// TIA Portal project "Drehgeber_0" (V20)

(* hardware
DEVICE "S7-1500/ET200MP-Station_1"  S7-1500 station
   slot 0: "Profilschiene_0"  Rack  6ES7 590-1***0-0AA0
   slot 1: "PLC_1"  CPU 1513-1 PN  6ES7 513-1AM03-0AB0  V4.0
      slot 3: "CPU-Display_1"  6ES7591-1AA00-0AA0
      slot 32768: "PROFINET-Schnittstelle_1"  X1
         slot 32769: "Port_1"  X1 P1
         slot 32770: "Port_2"  X1 P2
      slot 34817: "Virtual CP interface port_1"  Virtual CP interface port  Virtual CP interface port FW V4.0
   slot 2: "DI 16x24VDC BA_1"  DI 16x24VDC BA  6ES7 521-1BH10-0AA0  V1.1
   slot 3: "DQ 16x24VDC/0.5A ST_1"  DQ 16x24VDC/0.5A ST  6ES7 522-1BH00-0AB0  V2.0
   slot 4: "AI 8xU/I/R/RTD BA_2"  AI 8xU/I/R/RTD BA  6ES7 531-7QF00-0AB0  V1.0
   slot 5: "AQ 8xU/I HS_2"  AQ 8xU/I HS  6ES7 532-5HF00-0AB0  V2.2
*)

// ===== PLC "PLC_1"  CPU 1513-1 PN =====

VAR_GLOBAL   // PLC tag table "Eingaenge"
   "1B1" AT %I0.0 : Bool;   // Lichttaster
   "2B1" AT %I0.1 : Bool;   // Drehgeber (Signal A)
   "2B2" AT %I0.2 : Bool;   // Drehgeber (Signal B)
   "3B1" AT %E0.3 : Bool;   // Pusher 1 (hinten)
   "3B2" AT %E0.4 : Bool;   // Pusher 1 (vorne)
   "4B1" AT %E0.5 : Bool;   // Pusher 2 (hinten)
   "4B2" AT %E0.6 : Bool;   // Pusher 2 (vorne)
   "1B2" AT %ED30 : DInt;   // Sichtsensor
END_VAR

VAR_GLOBAL   // PLC tag table "Ausgaenge"
   "1M1" AT %Q0.1 : Bool;   // Förderband (vor)
   "1M2" AT %Q0.2 : Bool;   // Förderband (zurück)
   "3M1" AT %A0.3 : Bool;   // Pusher 1
   "4M1" AT %A0.5 : Bool;   // Pusher 2
END_VAR

DATA_BLOCK "Datenbaustein_1"   // DB1
{ S7_Optimized_Access := 'TRUE' }
VERSION : 0.1
   VAR
      Betriebsdaten : Struct
         Trigger : Struct
            Kanal_A : Struct
               Pos : Bool;
               Neg : Bool;
            END_STRUCT;
            Kanal_B : Struct
               Pos : Bool;
               Neg : Bool;
            END_STRUCT;
         END_STRUCT;
         Drehrichtung : Struct
            Vor : Bool;
            Zurueck : Bool;
         END_STRUCT;
         Pusher : Array[1..2] of Struct
            ID : UDInt;
            Pos_Register : DInt;
            Bauteil_Farbe : Array[0..1] of DInt;
            Zustand : Bool;
            PTRIG : Bool;
         END_STRUCT;
         Geberwert : DInt;
         Position_cm : Real;
         Schieben : Bool;
      END_STRUCT;
   END_VAR
BEGIN
   Betriebsdaten.Pusher[1].Pos_Register := 132;
   Betriebsdaten.Pusher[2].Pos_Register := 210;
END_DATA_BLOCK

DATA_BLOCK "Drehgeber_Signale_DB"   // DB2
{ S7_Optimized_Access := 'TRUE' }
VERSION : 0.1
// stored: InstanceOfName Drehgeber_Signale_Hohe_Aufloesung
"Drehgeber_Signale_Hohe_Aufloesung"
BEGIN
END_DATA_BLOCK

DATA_BLOCK "Schieberegister"   // DB3
{ S7_Optimized_Access := 'TRUE' }
VERSION : 0.1
   VAR
      Aktuelles_Bauteil : DInt;
      Register : Array[0..255] of DInt;
   END_VAR
BEGIN
END_DATA_BLOCK

FUNCTION_BLOCK "Drehgeber_Signale_Hohe_Aufloesung"   // FB1, FBD
{ S7_Optimized_Access := 'TRUE' }
VERSION : 0.1
   VAR
      Laufband_Richtung_DB : "Laufband_Richuntgserkennung";
   END_VAR
BEGIN

REGION Network 1
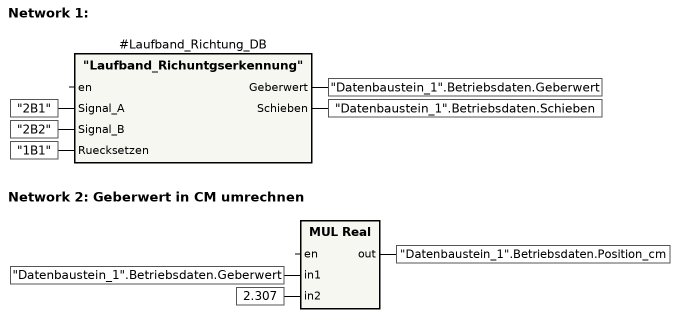
   #Laufband_Richtung_DB(Signal_A := "2B1",   // "Laufband_Richuntgserkennung"
                         Signal_B := "2B2",
                         Ruecksetzen := "1B1",
                         Geberwert => "Datenbaustein_1".Betriebsdaten.Geberwert,
                         Schieben => "Datenbaustein_1".Betriebsdaten.Schieben);
END_REGION

REGION Network 2: Geberwert in CM umrechnen
   "Datenbaustein_1".Betriebsdaten.Position_cm := "Datenbaustein_1".Betriebsdaten.Geberwert * 2.307;
END_REGION
END_FUNCTION_BLOCK

FUNCTION_BLOCK "Laufband_Richuntgserkennung"   // FB2, FBD
{ S7_Optimized_Access := 'TRUE' }
VERSION : 0.1
   VAR_INPUT
      Signal_A : Bool;
      Signal_B : Bool;
      Ruecksetzen : Bool;
   END_VAR
   VAR_OUTPUT
      Geberwert : DInt;
      Schieben : Bool;
   END_VAR
   VAR
      PTRIG_KanalA : Bool;
      NTRIG_KanalA : Bool;
      PTRIG_KanalB : Bool;
      NTRIG_KanalB : Bool;
      PTRIG_SignalA : Bool;
      PTRIG_SignalB : Bool;
      Vor : Bool;
      Zurueck : Bool;
   END_VAR
   VAR_TEMP   // added for the SCL form of the ladder/FBD networks
      _w1 : Bool;
      _w2 : Bool;
      _w3 : Bool;
      _w4 : Bool;
      _w5 : Bool;
   END_VAR
BEGIN

REGION Network 1: Vorwärts
   // Wenn eine positive Flanke von A kommt, wenn B bereits da ist = Vorwärts
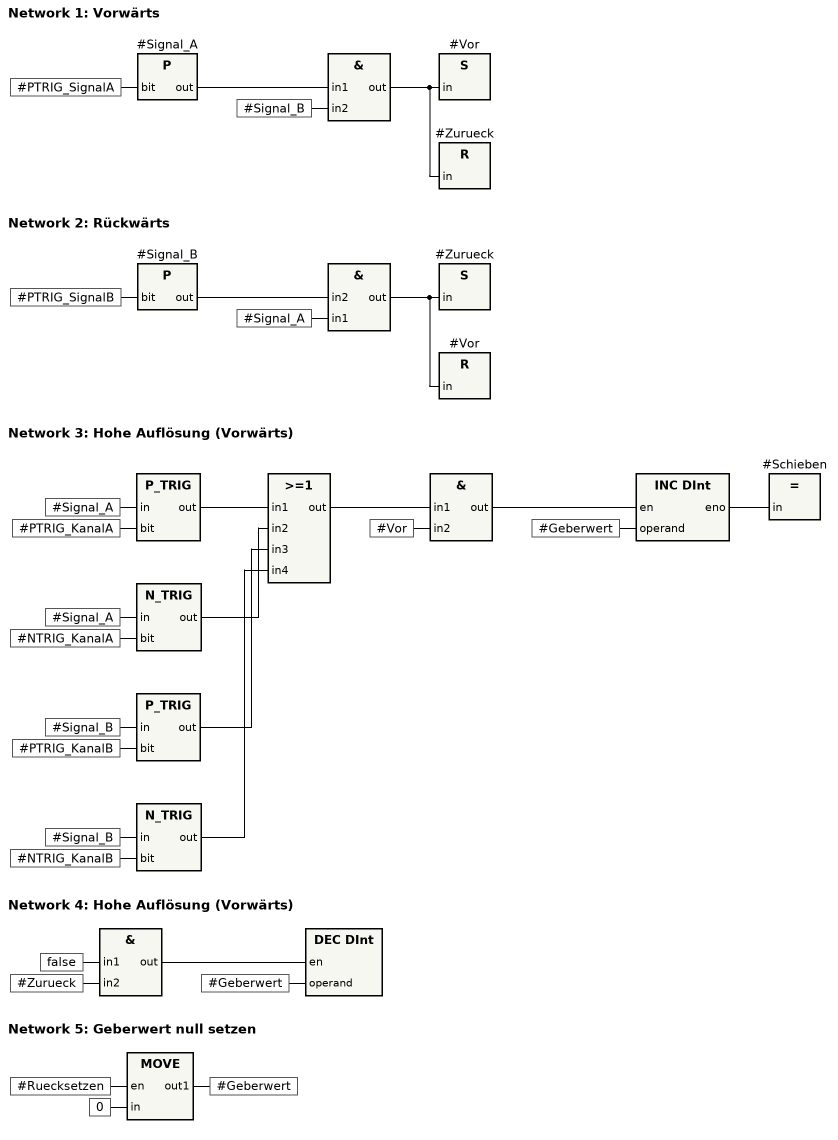
   #_w1 := #Signal_A AND NOT #PTRIG_SignalA;   // rising edge of #Signal_A
   #PTRIG_SignalA := #Signal_A;
   IF #_w1 AND #Signal_B THEN
       #Vor := TRUE;
       #Zurueck := FALSE;
   END_IF;
END_REGION

REGION Network 2: Rückwärts
   // Wenn eine positive Flanke von B kommt, wenn A bereits da ist = Rückwärts
   #_w1 := #Signal_B AND NOT #PTRIG_SignalB;   // rising edge of #Signal_B
   #PTRIG_SignalB := #Signal_B;
   IF #_w1 AND #Signal_A THEN
       #Zurueck := TRUE;
       #Vor := FALSE;
   END_IF;
END_REGION

REGION Network 3: Hohe Auflösung (Vorwärts)
   #_w1 := #Signal_A AND NOT #PTRIG_KanalA;   // rising edge
   #PTRIG_KanalA := #Signal_A;
   #_w2 := NOT #Signal_A AND #NTRIG_KanalA;   // falling edge
   #NTRIG_KanalA := #Signal_A;
   #_w3 := #Signal_B AND NOT #PTRIG_KanalB;   // rising edge
   #PTRIG_KanalB := #Signal_B;
   #_w4 := NOT #Signal_B AND #NTRIG_KanalB;   // falling edge
   #NTRIG_KanalB := #Signal_B;
   #_w5 := (#_w1 OR #_w2 OR #_w3 OR #_w4) AND #Vor;
   IF #_w5 THEN #Geberwert := #Geberwert + 1; END_IF;
   #Schieben := #_w5;
END_REGION

REGION Network 4: Hohe Auflösung (Vorwärts)
   IF false AND #Zurueck THEN #Geberwert := #Geberwert - 1; END_IF;
END_REGION

REGION Network 5: Geberwert null setzen
   IF #Ruecksetzen THEN #Geberwert := 0; END_IF;
END_REGION
END_FUNCTION_BLOCK

FUNCTION "Schieberegistersteuerung" : Void   // FC1, FBD
{ S7_Optimized_Access := 'TRUE' }
VERSION : 0.1
   VAR_INPUT
      Sensor_Ein : Bool;
      Vis_Sensor : DInt;
   END_VAR
   VAR_TEMP
      Iterator : DInt;
   END_VAR
BEGIN

REGION Network 1
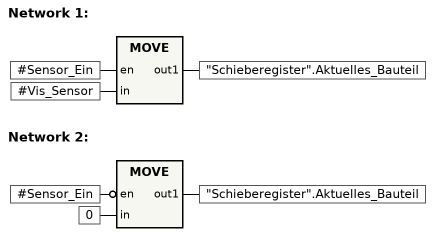
   IF #Sensor_Ein THEN "Schieberegister".Aktuelles_Bauteil := #Vis_Sensor; END_IF;
END_REGION

REGION Network 2
   IF NOT #Sensor_Ein THEN "Schieberegister".Aktuelles_Bauteil := 0; END_IF;
END_REGION

REGION Network 3 (SCL)
   //Wenn Signal vom Inkrementalgeber kommt, Register schieben
   IF "Datenbaustein_1".Betriebsdaten.Schieben THEN


       //.....dann For-Schleife ausführen
       FOR #Iterator := 250 TO 1 BY -1 DO
           "Schieberegister".Register[#Iterator] := "Schieberegister".Register[#Iterator - 1];
       END_FOR;

       //danach aktuellen Wert auf Register0
       "Schieberegister".Register[0] := "Schieberegister".Aktuelles_Bauteil;

   END_IF;
END_REGION
END_FUNCTION

FUNCTION "Pushersteuerung" : Void   // FC2, FBD
{ S7_Optimized_Access := 'TRUE' }
VERSION : 0.1
   VAR_INPUT
      Ausfahren : Bool;
      Einfahren : Bool;
   END_VAR
   VAR_OUTPUT
      Kolben : Bool;
   END_VAR
   VAR_IN_OUT
      Zustand : Bool;
   END_VAR
BEGIN

REGION Network 1
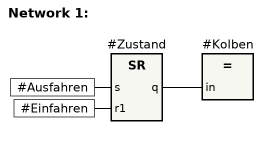
   IF #Ausfahren THEN
       #Zustand := TRUE;   // SR flip-flop
   END_IF;
   IF #Einfahren THEN #Zustand := FALSE; END_IF;
   #Kolben := #Zustand;
END_REGION
END_FUNCTION

FUNCTION "Pusher_Bauteil_schieben" : Void   // FC4, FBD
{ S7_Optimized_Access := 'TRUE' }
VERSION : 0.1
   VAR_INPUT
      Pusher_ID : DInt;
      Sensor_vorne : Bool;
   END_VAR
   VAR_OUTPUT
      Pusher_Motor : Bool;
   END_VAR
   VAR_TEMP
      Temp : Bool;
   END_VAR
   VAR_TEMP   // added for the SCL form of the ladder/FBD networks
      _w1 : Bool;
      _w2 : Bool;
   END_VAR
BEGIN

REGION Network 1
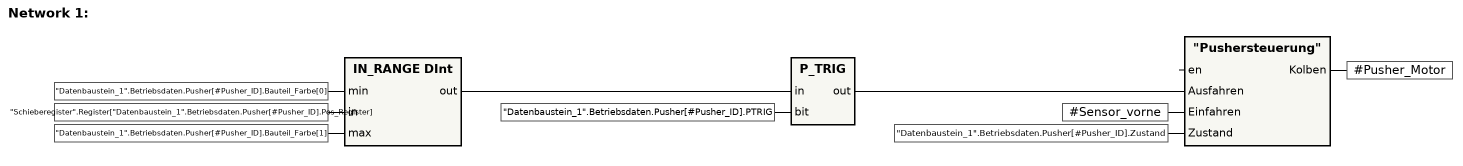
   #_w1 := ("Datenbaustein_1".Betriebsdaten.Pusher[#Pusher_ID].Bauteil_Farbe[0] <= "Schieberegister".Register["Datenbaustein_1".Betriebsdaten.Pusher[#Pusher_ID].Pos_Register]) AND ("Schieberegister".Register["Datenbaustein_1".Betriebsdaten.Pusher[#Pusher_ID].Pos_Register] <= "Datenbaustein_1".Betriebsdaten.Pusher[#Pusher_ID].Bauteil_Farbe[1]);
   #_w2 := #_w1 AND NOT "Datenbaustein_1".Betriebsdaten.Pusher[#Pusher_ID].PTRIG;   // rising edge
   "Datenbaustein_1".Betriebsdaten.Pusher[#Pusher_ID].PTRIG := #_w1;
   "Pushersteuerung"(Ausfahren := #_w2,
                     Einfahren := #Sensor_vorne,
                     Zustand := "Datenbaustein_1".Betriebsdaten.Pusher[#Pusher_ID].Zustand,
                     Kolben => #Pusher_Motor);
END_REGION
END_FUNCTION

ORGANIZATION_BLOCK "Main"   // OB1, FBD, ProgramCycle
TITLE = "Main Program Sweep (Cycle)"
{ S7_Optimized_Access := 'TRUE' }
VERSION : 0.1
   VAR_INPUT
      Initial_Call : Bool;   // Initial call of this OB
      Remanence : Bool;   // =True, if remanent data are available
   END_VAR
BEGIN

REGION Network 1
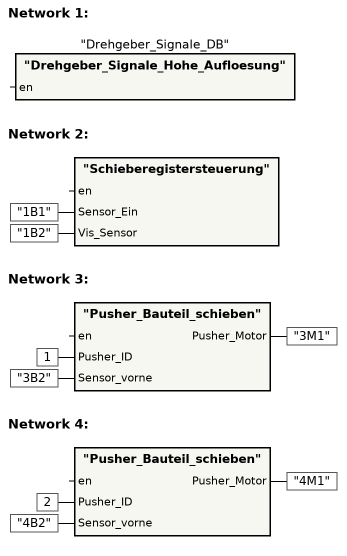
   "Drehgeber_Signale_DB"();   // "Drehgeber_Signale_Hohe_Aufloesung"
END_REGION

REGION Network 2
   "Schieberegistersteuerung"(Sensor_Ein := "1B1", Vis_Sensor := "1B2");
END_REGION

REGION Network 3
   "Pusher_Bauteil_schieben"(Pusher_ID := 1, Sensor_vorne := "3B2", Pusher_Motor => "3M1");
END_REGION

REGION Network 4
   "Pusher_Bauteil_schieben"(Pusher_ID := 2, Sensor_vorne := "4B2", Pusher_Motor => "4M1");
END_REGION
END_ORGANIZATION_BLOCK